FUNCTION_BLOCK PAEActSlider EXTENDS PAEActuator1way
VAR_INPUT
END_VAR
VAR_OUTPUT
END_VAR
VAR
END_VAR

END_FUNCTION_BLOCK

(* stored: Version 1.1.0.1, ProductVersion 3.1.4020.12
   POU PAEActSlider: Id {0512d245-df30-415f-b9ad-faab750d638c}, SpecialFunc None *)
